FUNCTION_BLOCK FB_SensorBase EXTENDS FB_Device
VAR_INPUT
END_VAR
VAR_OUTPUT
END_VAR
VAR
END_VAR

METHOD  HandleMessage : BOOL
VAR_INPUT
	message :STRING;
END_VAR
END_METHOD

END_FUNCTION_BLOCK

(* stored: Version 1.1.0.1, ProductVersion 3.1.4024.9
   POU FB_SensorBase: Id {7f3b2266-956f-4033-aaea-f3c25f958529}, SpecialFunc None
   Method HandleMessage: Id {402cfd41-6c77-4bd5-aafc-0d7a618f5f85} *)
